(* PLC project Unnamed, Unknown Unnamed 1 *)
(* stored: creationDateTime 2022-02-28T03:29:20, modificationDateTime 2022-03-29T14:34:43 *)

PROGRAM program0
  VAR
    LocalVar0 : BOOL;
    LocalVar1 : BOOL;
    LocalVar2 : BOOL;
    LocalVar3 : BOOL;
    LocalVar4 : BOOL;
  END_VAR

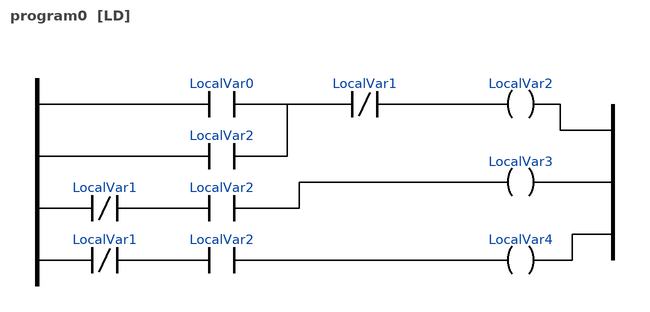
(* LD diagram, written out as Structured Text *)
LocalVar2 := (LocalVar0 OR LocalVar2) AND NOT LocalVar1;
LocalVar3 := NOT LocalVar1 AND LocalVar2;
LocalVar4 := NOT LocalVar1 AND LocalVar2;
END_PROGRAM

CONFIGURATION Config0
  RESOURCE Res0 ON PLC
    TASK task0(INTERVAL := T#20ms, PRIORITY := 0);
    PROGRAM instance0 WITH task0 : program0;
  END_RESOURCE
END_CONFIGURATION
